FUNCTION F_BarToPascal : LREAL
VAR_INPUT
	fBar : LREAL;
END_VAR
VAR
END_VAR

F_BarToPascal := fBar*1E5;

END_FUNCTION

(* stored: Version 1.1.0.1, ProductVersion 3.1.4024.10
   POU F_BarToPascal: Id {587ec4da-2a67-498f-936b-937080727254}, SpecialFunc None *)
